// TIA Portal V16 export
// export: Created 2023-03-29T11:04:48.8818809Z, ExportSetting WithDefaults, DisplayName Totally Integrated Automation Portal, DisplayVersion V16 Update 6, DisplayName TIA Portal Version Control Interface, DisplayVersion V16 Update 2, DisplayName TIA Portal Openness, DisplayVersion V16 Update 6, DisplayName STEP 7 Professional, DisplayVersion V16 Update 6, DisplayName STEP 7 Safety, DisplayVersion V16, DisplayName WinCC Advanced, DisplayVersion V16 Update 6
FUNCTION_BLOCK "Sterowanie falownikiem"   // FB11, LAD
TITLE = Control of Inverters
{ S7_Optimized_Access := 'TRUE' }
AUTHOR : rtecmer
VERSION : 0.1
// Sterowanie przekaćnikiem załączającym falownik do pracy
// stored: AutoNumber true, IsIECCheckEnabled false, IsRetainMemResEnabled false, MemoryReserve 500, SetENOAutomatically false, UDAEnableTagReadback false
   VAR_INPUT
      IsModeAut : Bool;   // Znacznik tryb automat dla pomp
      AlwaysTRUE : Bool;
      Set_HWork_P1 : Bool;   // Znacznik ustawienia pracy od licznika pracy
      Set_HWork_P2 : Bool;   // Znacznik ustawienia pracy od licznika pracy
      Set_HWork_P3 : Bool;   // Znacznik ustawienia pracy od licznika pracy
      Set_HWork_P4 : Bool;
      setPID_Pomp : Bool;   // Znacznik załączenie, regulacji falownika
      Is_loading_K3 : Bool;   // Znacznik pompy wiodącej
      IsRunInverter_P4 : Bool;
      IsRunInverter_P3 : Bool;   // Potwierdzenie załączenie stycznika falownik pompy
      IsRunInverter_P2 : Bool;   // Potwierdzenie załączenie stycznika falownik pompy
      IsRunInverter_P1 : Bool;   // Potwierdzenie załączenie stycznika falownik pompy
      Bit_Aut_P1 : Bool;   // Bit tryb prac automat
      Bit_Aut_P2 : Bool;   // Bit tryb prac automat
      Bit_Aut_P3 : Bool;   // Bit tryb prac automat
      Bit_Aut_P4 : Bool;
      IsRunNetwork_P1 : Bool;   // Potwierdzenie załączenie stycznika sieć
      IsRunNetwork_P2 : Bool := false;   // Potwierdzenie załączenie stycznika sieć
      IsRunNetwork_P3 : Bool := false;   // Potwierdzenie załączenie stycznika sieć
      IsRunNetwork_P4 : Bool;
   END_VAR
   VAR_OUTPUT
      CMD_start_stop_inverter : Bool;   // Przekaźnik sterowania załączaniem falownika
   END_VAR
   VAR
      Res_upHz : Bool;   // Reset znacznika up_Hz wyłaczenie dodatkowe
   END_VAR
BEGIN

REGION Network 1: Reset bitu pomocniczego ustalenia przyrostu Hz
   // Kasowanie podczas rozruchu po restarcie
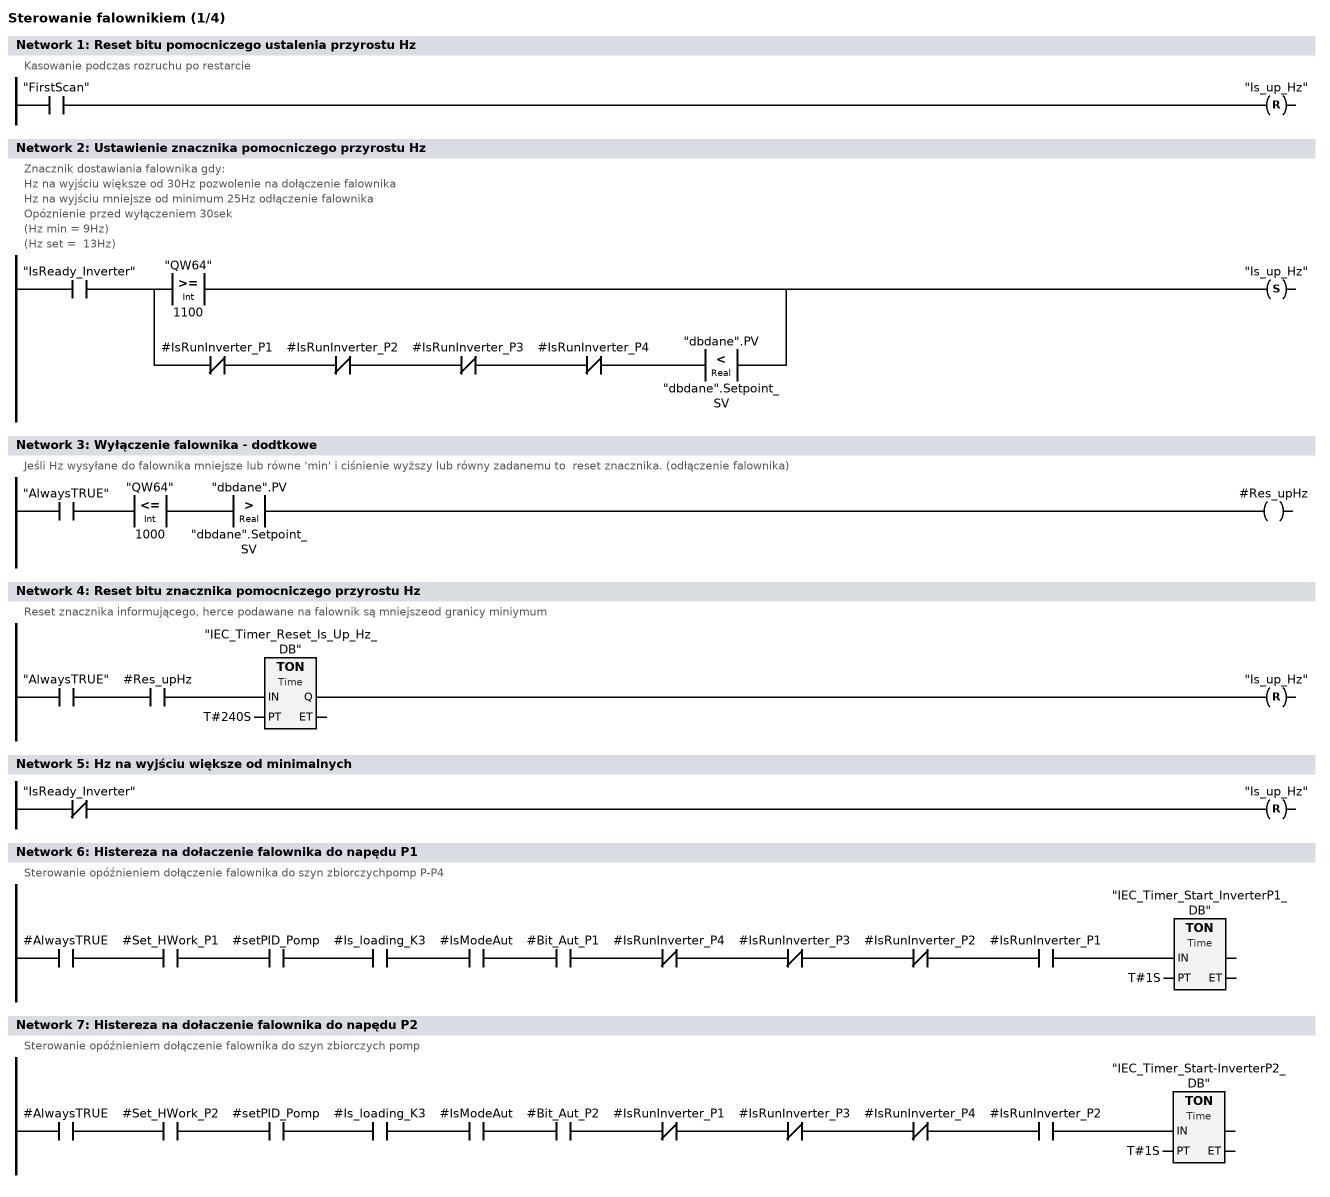
   RUNG wire#powerrail
      Contact( "FirstScan" )
      R_Coil( "Is_up_Hz" )
   END_RUNG
   // the same network as SCL:
   IF "FirstScan" THEN "Is_up_Hz" := FALSE; END_IF;
END_REGION

REGION Network 2: Ustawienie znacznika pomocniczego przyrostu Hz
   // Znacznik dostawiania falownika gdy:
   // Hz na wyjściu większe od 30Hz pozwolenie na dołączenie falownika
   // Hz na wyjściu mniejsze od minimum 25Hz odłączenie falownika
   // Opóznienie przed wyłączeniem 30sek
   // (Hz min = 9Hz)
   // (Hz set =  13Hz)
   RUNG wire#powerrail
      Contact( "IsReady_Inverter" )
      wire#w1
      { S7_Templates := "SrcType := Int" } GE_Contact(in1 := "QW64", in2 := 1100)
      wire#w2
      S_Coil( "Is_up_Hz" )
   END_RUNG
   RUNG wire#w1
      I_Contact( #IsRunInverter_P1 )
      I_Contact( #IsRunInverter_P2 )
      I_Contact( #IsRunInverter_P3 )
      I_Contact( #IsRunInverter_P4 )
      { S7_Templates := "SrcType := Real" } LT_Contact(in1 := "dbdane".PV, in2 := "dbdane".Setpoint_SV)
   END_RUNG wire#w2
   // the same network as SCL:
   IF "IsReady_Inverter" AND (("QW64" >= 1100) OR (NOT #IsRunInverter_P1 AND NOT #IsRunInverter_P2 AND NOT #IsRunInverter_P3 AND NOT #IsRunInverter_P4 AND ("dbdane".PV < "dbdane".Setpoint_SV))) THEN
       "Is_up_Hz" := TRUE;
   END_IF;
END_REGION

REGION Network 3: Wyłączenie falownika - dodtkowe
   // Jeśli Hz wysyłane do falownika mniejsze lub równe 'min' i ciśnienie wyższy lub równy zadanemu to  reset znacznika. (odłączenie falownika)
   RUNG wire#powerrail
      Contact( "AlwaysTRUE" )
      { S7_Templates := "SrcType := Int" } LE_Contact(in1 := "QW64", in2 := 1000)
      { S7_Templates := "SrcType := Real" } GT_Contact(in1 := "dbdane".PV, in2 := "dbdane".Setpoint_SV)
      Coil( #Res_upHz )
   END_RUNG
   // the same network as SCL:
   #Res_upHz := "AlwaysTRUE" AND ("QW64" <= 1000) AND ("dbdane".PV > "dbdane".Setpoint_SV);
END_REGION

REGION Network 4: Reset bitu znacznika pomocniczego przyrostu Hz
   // Reset znacznika informującego, herce podawane na falownik są mniejszeod granicy miniymum
   RUNG wire#powerrail
      Contact( "AlwaysTRUE" )
      Contact( #Res_upHz )
      { S7_Templates := "time_type := Time" } "IEC_Timer_Reset_Is_Up_Hz_DB".TON(pt := T#240S, et =>)
      R_Coil( "Is_up_Hz" )
   END_RUNG
   // the same network as SCL:
   "IEC_Timer_Reset_Is_Up_Hz_DB".TON(IN := "AlwaysTRUE" AND #Res_upHz, PT := T#240S);
   IF "IEC_Timer_Reset_Is_Up_Hz_DB".Q THEN "Is_up_Hz" := FALSE; END_IF;
END_REGION

REGION Network 5: Hz na wyjściu większe od minimalnych
   RUNG wire#powerrail
      I_Contact( "IsReady_Inverter" )
      R_Coil( "Is_up_Hz" )
   END_RUNG
   // the same network as SCL:
   IF NOT "IsReady_Inverter" THEN "Is_up_Hz" := FALSE; END_IF;
END_REGION

REGION Network 6: Histereza na dołaczenie falownika do napędu P1
   // Sterowanie opóźnieniem dołączenie falownika do szyn zbiorczychpomp P-P4
   RUNG wire#powerrail
      Contact( #AlwaysTRUE )
      Contact( #Set_HWork_P1 )
      Contact( #setPID_Pomp )
      Contact( #Is_loading_K3 )
      Contact( #IsModeAut )
      Contact( #Bit_Aut_P1 )
      I_Contact( #IsRunInverter_P4 )
      I_Contact( #IsRunInverter_P3 )
      I_Contact( #IsRunInverter_P2 )
      Contact( #IsRunInverter_P1 )
      { S7_Templates := "time_type := Time" } "IEC_Timer_Start_InverterP1_DB".TON(pt := T#1S, et =>)
   END_RUNG
   // the same network as SCL:
   "IEC_Timer_Start_InverterP1_DB".TON(IN := #AlwaysTRUE AND #Set_HWork_P1 AND #setPID_Pomp AND #Is_loading_K3 AND #IsModeAut AND #Bit_Aut_P1 AND NOT #IsRunInverter_P4 AND NOT #IsRunInverter_P3 AND NOT #IsRunInverter_P2 AND #IsRunInverter_P1,
                           PT := T#1S);
END_REGION

REGION Network 7: Histereza na dołaczenie falownika do napędu P2
   // Sterowanie opóźnieniem dołączenie falownika do szyn zbiorczych pomp
   RUNG wire#powerrail
      Contact( #AlwaysTRUE )
      Contact( #Set_HWork_P2 )
      Contact( #setPID_Pomp )
      Contact( #Is_loading_K3 )
      Contact( #IsModeAut )
      Contact( #Bit_Aut_P2 )
      I_Contact( #IsRunInverter_P1 )
      I_Contact( #IsRunInverter_P3 )
      I_Contact( #IsRunInverter_P4 )
      Contact( #IsRunInverter_P2 )
      { S7_Templates := "time_type := Time" } "IEC_Timer_Start-InverterP2_DB".TON(pt := T#1S, et =>)
   END_RUNG
   // the same network as SCL:
   "IEC_Timer_Start-InverterP2_DB".TON(IN := #AlwaysTRUE AND #Set_HWork_P2 AND #setPID_Pomp AND #Is_loading_K3 AND #IsModeAut AND #Bit_Aut_P2 AND NOT #IsRunInverter_P1 AND NOT #IsRunInverter_P3 AND NOT #IsRunInverter_P4 AND #IsRunInverter_P2,
                           PT := T#1S);
END_REGION

REGION Network 8: Histereza na dołaczenie falownika do napędu P3
   // Sterowanie opóźnieniem dołączenie falownika do szyn zbiorczych kompresorów
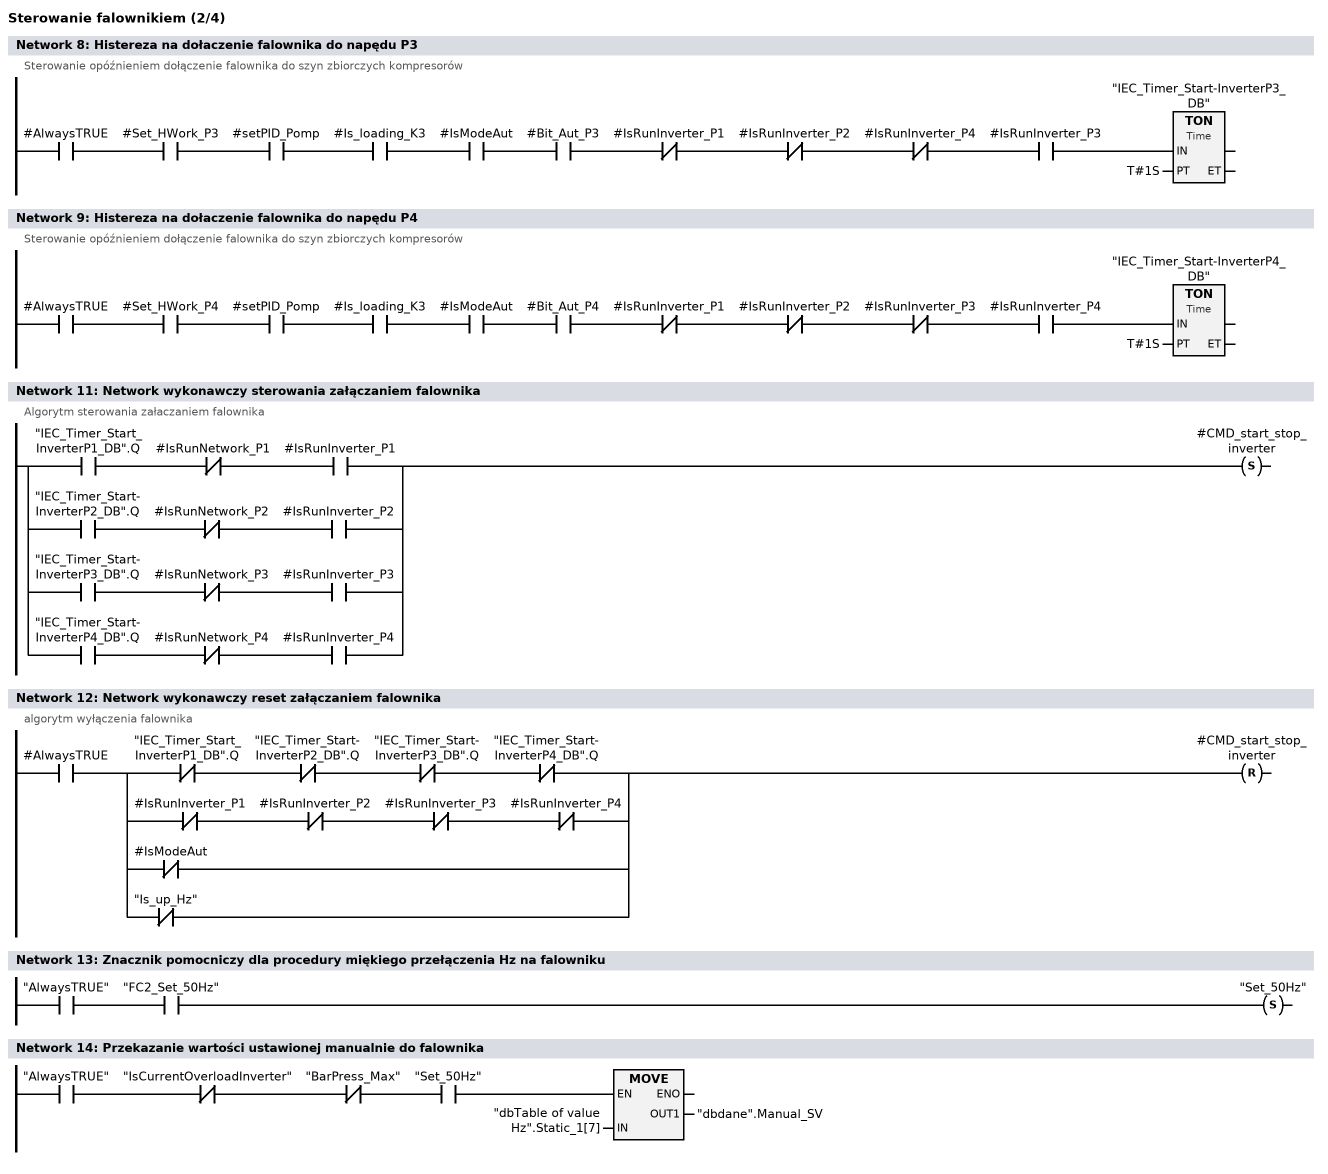
   RUNG wire#powerrail
      Contact( #AlwaysTRUE )
      Contact( #Set_HWork_P3 )
      Contact( #setPID_Pomp )
      Contact( #Is_loading_K3 )
      Contact( #IsModeAut )
      Contact( #Bit_Aut_P3 )
      I_Contact( #IsRunInverter_P1 )
      I_Contact( #IsRunInverter_P2 )
      I_Contact( #IsRunInverter_P4 )
      Contact( #IsRunInverter_P3 )
      { S7_Templates := "time_type := Time" } "IEC_Timer_Start-InverterP3_DB".TON(pt := T#1S, et =>)
   END_RUNG
   // the same network as SCL:
   "IEC_Timer_Start-InverterP3_DB".TON(IN := #AlwaysTRUE AND #Set_HWork_P3 AND #setPID_Pomp AND #Is_loading_K3 AND #IsModeAut AND #Bit_Aut_P3 AND NOT #IsRunInverter_P1 AND NOT #IsRunInverter_P2 AND NOT #IsRunInverter_P4 AND #IsRunInverter_P3,
                           PT := T#1S);
END_REGION

REGION Network 9: Histereza na dołaczenie falownika do napędu P4
   // Sterowanie opóźnieniem dołączenie falownika do szyn zbiorczych kompresorów
   RUNG wire#powerrail
      Contact( #AlwaysTRUE )
      Contact( #Set_HWork_P4 )
      Contact( #setPID_Pomp )
      Contact( #Is_loading_K3 )
      Contact( #IsModeAut )
      Contact( #Bit_Aut_P4 )
      I_Contact( #IsRunInverter_P1 )
      I_Contact( #IsRunInverter_P2 )
      I_Contact( #IsRunInverter_P3 )
      Contact( #IsRunInverter_P4 )
      { S7_Templates := "time_type := Time" } "IEC_Timer_Start-InverterP4_DB".TON(pt := T#1S, et =>)
   END_RUNG
   // the same network as SCL:
   "IEC_Timer_Start-InverterP4_DB".TON(IN := #AlwaysTRUE AND #Set_HWork_P4 AND #setPID_Pomp AND #Is_loading_K3 AND #IsModeAut AND #Bit_Aut_P4 AND NOT #IsRunInverter_P1 AND NOT #IsRunInverter_P2 AND NOT #IsRunInverter_P3 AND #IsRunInverter_P4,
                           PT := T#1S);
END_REGION

REGION Network 11: Network wykonawczy sterowania załączaniem falownika
   // Algorytm sterowania załaczaniem falownika
   RUNG wire#powerrail
      Contact( "IEC_Timer_Start_InverterP1_DB".Q )
      I_Contact( #IsRunNetwork_P1 )
      Contact( #IsRunInverter_P1 )
      wire#w1
      S_Coil( #CMD_start_stop_inverter )
   END_RUNG
   RUNG wire#powerrail
      Contact( "IEC_Timer_Start-InverterP2_DB".Q )
      I_Contact( #IsRunNetwork_P2 )
      Contact( #IsRunInverter_P2 )
   END_RUNG wire#w1
   RUNG wire#powerrail
      Contact( "IEC_Timer_Start-InverterP3_DB".Q )
      I_Contact( #IsRunNetwork_P3 )
      Contact( #IsRunInverter_P3 )
   END_RUNG wire#w1
   RUNG wire#powerrail
      Contact( "IEC_Timer_Start-InverterP4_DB".Q )
      I_Contact( #IsRunNetwork_P4 )
      Contact( #IsRunInverter_P4 )
   END_RUNG wire#w1
   // the same network as SCL:
   IF ("IEC_Timer_Start_InverterP1_DB".Q AND NOT #IsRunNetwork_P1 AND #IsRunInverter_P1) OR ("IEC_Timer_Start-InverterP2_DB".Q AND NOT #IsRunNetwork_P2 AND #IsRunInverter_P2) OR ("IEC_Timer_Start-InverterP3_DB".Q AND NOT #IsRunNetwork_P3 AND #IsRunInverter_P3) OR ("IEC_Timer_Start-InverterP4_DB".Q AND NOT #IsRunNetwork_P4 AND #IsRunInverter_P4) THEN
       #CMD_start_stop_inverter := TRUE;
   END_IF;
END_REGION

REGION Network 12: Network wykonawczy reset załączaniem falownika
   // algorytm wyłączenia falownika
   RUNG wire#powerrail
      Contact( #AlwaysTRUE )
      wire#w1
      I_Contact( "IEC_Timer_Start_InverterP1_DB".Q )
      I_Contact( "IEC_Timer_Start-InverterP2_DB".Q )
      I_Contact( "IEC_Timer_Start-InverterP3_DB".Q )
      I_Contact( "IEC_Timer_Start-InverterP4_DB".Q )
      wire#w2
      R_Coil( #CMD_start_stop_inverter )
   END_RUNG
   RUNG wire#w1
      I_Contact( #IsRunInverter_P1 )
      I_Contact( #IsRunInverter_P2 )
      I_Contact( #IsRunInverter_P3 )
      I_Contact( #IsRunInverter_P4 )
   END_RUNG wire#w2
   RUNG wire#w1
      I_Contact( #IsModeAut )
   END_RUNG wire#w2
   RUNG wire#w1
      I_Contact( "Is_up_Hz" )
   END_RUNG wire#w2
   // the same network as SCL:
   IF #AlwaysTRUE AND ((NOT "IEC_Timer_Start_InverterP1_DB".Q AND NOT "IEC_Timer_Start-InverterP2_DB".Q AND NOT "IEC_Timer_Start-InverterP3_DB".Q AND NOT "IEC_Timer_Start-InverterP4_DB".Q) OR (NOT #IsRunInverter_P1 AND NOT #IsRunInverter_P2 AND NOT #IsRunInverter_P3 AND NOT #IsRunInverter_P4) OR NOT #IsModeAut OR NOT "Is_up_Hz") THEN
       #CMD_start_stop_inverter := FALSE;
   END_IF;
END_REGION

REGION Network 13: Znacznik pomocniczy dla procedury miękiego przełączenia Hz na falowniku
   RUNG wire#powerrail
      Contact( "AlwaysTRUE" )
      Contact( "FC2_Set_50Hz" )
      S_Coil( "Set_50Hz" )
   END_RUNG
   // the same network as SCL:
   IF "AlwaysTRUE" AND "FC2_Set_50Hz" THEN "Set_50Hz" := TRUE; END_IF;
END_REGION

REGION Network 14: Przekazanie wartości ustawionej manualnie do falownika
   RUNG wire#powerrail
      Contact( "AlwaysTRUE" )
      I_Contact( "IsCurrentOverloadInverter" )
      I_Contact( "BarPress_Max" )
      Contact( "Set_50Hz" )
      Move(in := "dbTable of value Hz".Static_1[7], out1 => "dbdane".Manual_SV)
   END_RUNG
   // the same network as SCL:
   IF "AlwaysTRUE" AND NOT "IsCurrentOverloadInverter" AND NOT "BarPress_Max" AND "Set_50Hz" THEN
       "dbdane".Manual_SV := "dbTable of value Hz".Static_1[7];
   END_IF;
END_REGION

REGION Network 15: Przekazanie wartości ustawionej manualnie do falownika gdy awaria max ciśnienie
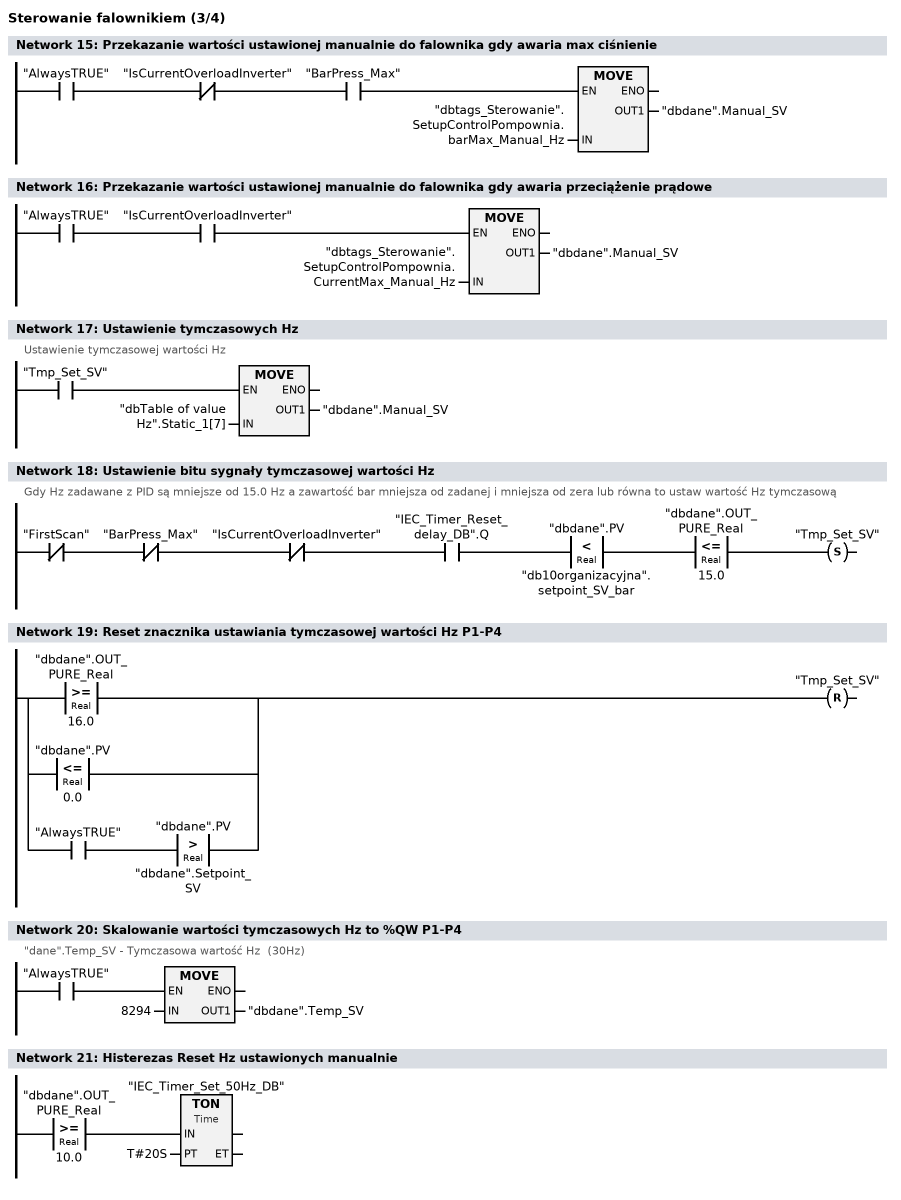
   RUNG wire#powerrail
      Contact( "AlwaysTRUE" )
      I_Contact( "IsCurrentOverloadInverter" )
      Contact( "BarPress_Max" )
      Move(in := "dbtags_Sterowanie".SetupControlPompownia.barMax_Manual_Hz, out1 => "dbdane".Manual_SV)
   END_RUNG
   // the same network as SCL:
   IF "AlwaysTRUE" AND NOT "IsCurrentOverloadInverter" AND "BarPress_Max" THEN
       "dbdane".Manual_SV := "dbtags_Sterowanie".SetupControlPompownia.barMax_Manual_Hz;
   END_IF;
END_REGION

REGION Network 16: Przekazanie wartości ustawionej manualnie do falownika gdy awaria przeciążenie prądowe
   RUNG wire#powerrail
      Contact( "AlwaysTRUE" )
      Contact( "IsCurrentOverloadInverter" )
      Move(in := "dbtags_Sterowanie".SetupControlPompownia.CurrentMax_Manual_Hz, out1 => "dbdane".Manual_SV)
   END_RUNG
   // the same network as SCL:
   IF "AlwaysTRUE" AND "IsCurrentOverloadInverter" THEN
       "dbdane".Manual_SV := "dbtags_Sterowanie".SetupControlPompownia.CurrentMax_Manual_Hz;
   END_IF;
END_REGION

REGION Network 17: Ustawienie tymczasowych Hz
   // Ustawienie tymczasowej wartości Hz
   RUNG wire#powerrail
      Contact( "Tmp_Set_SV" )
      Move(in := "dbTable of value Hz".Static_1[7], out1 => "dbdane".Manual_SV)
   END_RUNG
   // the same network as SCL:
   IF "Tmp_Set_SV" THEN "dbdane".Manual_SV := "dbTable of value Hz".Static_1[7]; END_IF;
END_REGION

REGION Network 18: Ustawienie bitu sygnały tymczasowej wartości Hz
   // Gdy Hz zadawane z PID są mniejsze od 15.0 Hz a zawartość bar mniejsza od zadanej i mniejsza od zera lub równa to ustaw wartość Hz tymczasową
   RUNG wire#powerrail
      I_Contact( "FirstScan" )
      I_Contact( "BarPress_Max" )
      I_Contact( "IsCurrentOverloadInverter" )
      Contact( "IEC_Timer_Reset_delay_DB".Q )
      { S7_Templates := "SrcType := Real" } LT_Contact(in1 := "dbdane".PV, in2 := "db10organizacyjna".setpoint_SV_bar)
      { S7_Templates := "SrcType := Real" } LE_Contact(in1 := "dbdane".OUT_PURE_Real, in2 := 15.0)
      S_Coil( "Tmp_Set_SV" )
   END_RUNG
   // the same network as SCL:
   IF NOT "FirstScan" AND NOT "BarPress_Max" AND NOT "IsCurrentOverloadInverter" AND "IEC_Timer_Reset_delay_DB".Q AND ("dbdane".PV < "db10organizacyjna".setpoint_SV_bar) AND ("dbdane".OUT_PURE_Real <= 15.0) THEN
       "Tmp_Set_SV" := TRUE;
   END_IF;
END_REGION

REGION Network 19: Reset znacznika ustawiania tymczasowej wartości Hz P1-P4
   RUNG wire#powerrail
      { S7_Templates := "SrcType := Real" } GE_Contact(in1 := "dbdane".OUT_PURE_Real, in2 := 16.0)
      wire#w1
      R_Coil( "Tmp_Set_SV" )
   END_RUNG
   RUNG wire#powerrail
      { S7_Templates := "SrcType := Real" } LE_Contact(in1 := "dbdane".PV, in2 := 0.0)
   END_RUNG wire#w1
   RUNG wire#powerrail
      Contact( "AlwaysTRUE" )
      { S7_Templates := "SrcType := Real" } GT_Contact(in1 := "dbdane".PV, in2 := "dbdane".Setpoint_SV)
   END_RUNG wire#w1
   // the same network as SCL:
   IF ("dbdane".OUT_PURE_Real >= 16.0) OR ("dbdane".PV <= 0.0) OR ("AlwaysTRUE" AND ("dbdane".PV > "dbdane".Setpoint_SV)) THEN
       "Tmp_Set_SV" := FALSE;
   END_IF;
END_REGION

REGION Network 20: Skalowanie wartości tymczasowych Hz to %QW P1-P4
   // "dane".Temp_SV - Tymczasowa wartość Hz  (30Hz)
   RUNG wire#powerrail
      Contact( "AlwaysTRUE" )
      Move(in := 8294, out1 => "dbdane".Temp_SV)
   END_RUNG
   // the same network as SCL:
   IF "AlwaysTRUE" THEN "dbdane".Temp_SV := 8294; END_IF;
END_REGION

REGION Network 21: Histerezas Reset Hz ustawionych manualnie
   RUNG wire#powerrail
      { S7_Templates := "SrcType := Real" } GE_Contact(in1 := "dbdane".OUT_PURE_Real, in2 := 10.0)
      { S7_Templates := "time_type := Time" } "IEC_Timer_Set_50Hz_DB".TON(pt := T#20S, et =>)
   END_RUNG
   // the same network as SCL:
   "IEC_Timer_Set_50Hz_DB".TON(IN := "dbdane".OUT_PURE_Real >= 10.0, PT := T#20S);
END_REGION

REGION Network 22: Reset znacznika płynnego przełaczenie Hz z tymczasowych na podawane z PID
   // Reset znacznika manualnego zadawania Hz
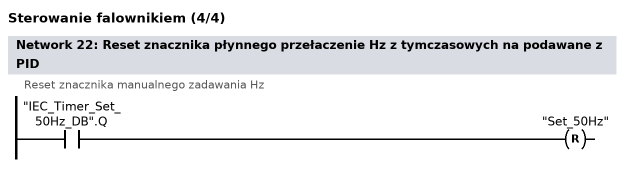
   RUNG wire#powerrail
      Contact( "IEC_Timer_Set_50Hz_DB".Q )
      R_Coil( "Set_50Hz" )
   END_RUNG
   // the same network as SCL:
   IF "IEC_Timer_Set_50Hz_DB".Q THEN "Set_50Hz" := FALSE; END_IF;
END_REGION
END_FUNCTION_BLOCK
